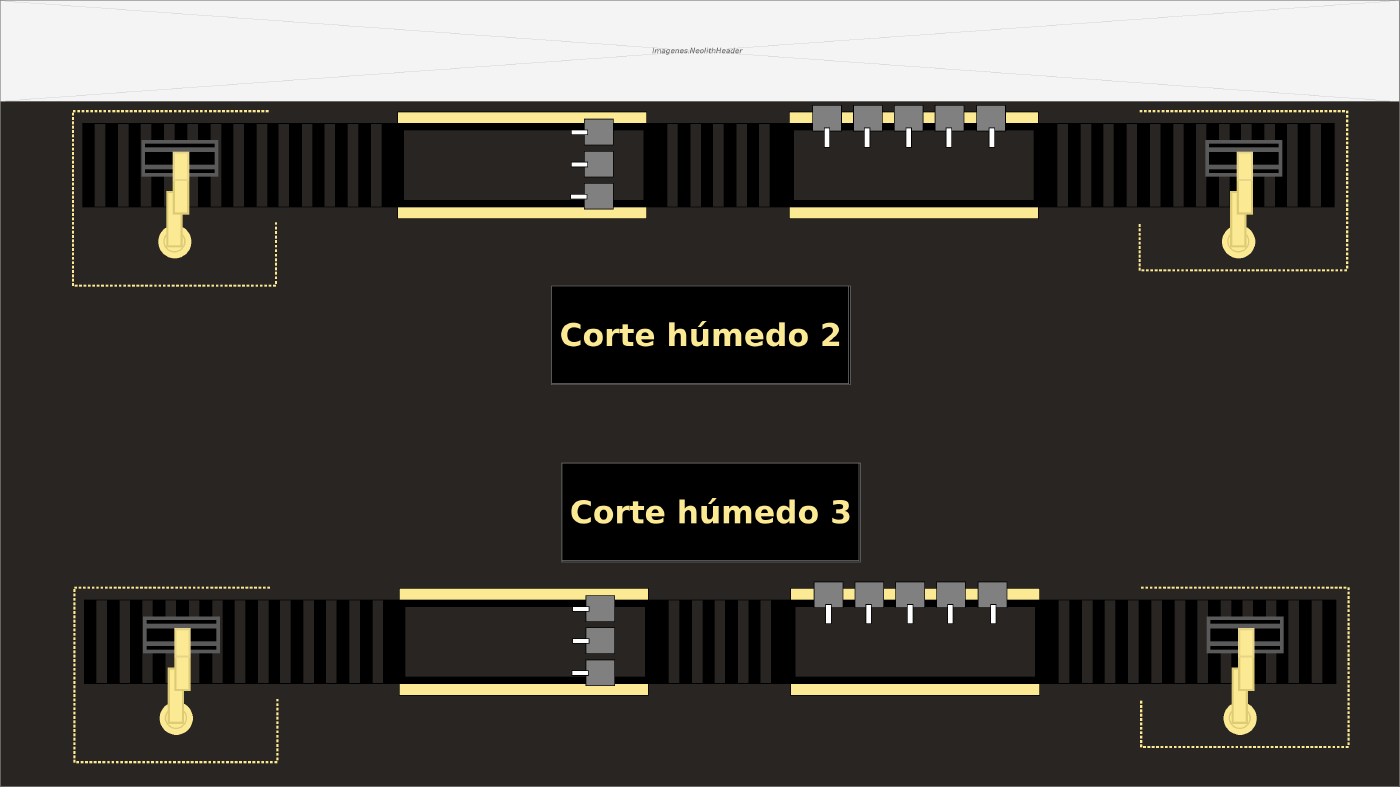
VISUALIZATION Home_Sel_Maq  // 1920x1080
    Button (756,392 410x136), "Corte húmedo 2"
        OnMouseUp: change screen: Home_CortH2
    Button (770,635 410x136), "Corte húmedo 3"
        OnMouseUp: change screen: Home_CortH3
    Image (-7,0 1927x139), image: Imagenes.NeolithHeader
    Group (100,144 1747x248)
        Rectangle (445,9 342x147)
        Rectangle (982,9 342x147)
        Rectangle (13,25 1717x115)
        Group (1349,25 363x115)
            Rectangle (0,0 16x115)
            Rectangle (32,0 16x115)
            Group (63,0 48x115)
                Rectangle (0,0 16x115)
                Rectangle (32,0 16x115)
            Group (127,0 111x115)
                Rectangle (0,0 16x115)
                Rectangle (32,0 16x115)
                Group (63,0 48x115)
                    Rectangle (0,0 16x115)
                    Rectangle (32,0 16x115)
            Rectangle (252,0 16x115)
            Rectangle (284,0 16x115)
            Group (315,0 48x115)
                Rectangle (0,0 16x115)
                Rectangle (32,0 16x115)
        Group (29,25 363x115)
            Rectangle (0,0 16x115)
            Rectangle (32,0 16x115)
            Group (63,0 48x115)
                Rectangle (0,0 16x115)
                Rectangle (32,0 16x115)
            Group (127,0 111x115)
                Rectangle (0,0 16x115)
                Rectangle (32,0 16x115)
                Group (63,0 48x115)
                    Rectangle (0,0 16x115)
                    Rectangle (32,0 16x115)
            Rectangle (252,0 16x115)
            Rectangle (284,0 16x115)
            Group (315,0 48x115)
                Rectangle (0,0 16x115)
                Rectangle (32,0 16x115)
        Rectangle (408,25 16x115)
        Rectangle (453,34 330x97)
        Rectangle (701,19 40x36)
        Rectangle (701,63 40x36)
        Rectangle (701,107 40x36)
        Rectangle (683,34 23x7)
        Rectangle (683,78 23x7)
        Rectangle (682,122 23x7)
        Rectangle (988,34 330x97)
        Rectangle (1014,0 40x36)
        Rectangle (1070,0 40x36)
        Rectangle (1126,0 40x36)
        Rectangle (1182,0 40x36)
        Rectangle (1239,0 40x36)
        Rectangle (1085,31 8x27)
        Rectangle (1030,31 8x27)
        Rectangle (1142,31 8x27)
        Rectangle (1197,31 8x27)
        Rectangle (1256,31 8x27)
        Group (814,25 142x115)
            Rectangle (126,0 16x115)
            Rectangle (0,0 16x115)
            Rectangle (32,0 16x115)
            Group (63,0 48x115)
                Rectangle (0,0 16x115)
                Rectangle (32,0 16x115)
        Polyline (1463,8) (1747,8) (1747,227) (1463,227) (1463,161)
        Polyline (278,161) (278,248) (0,248) (0,8) (271,8)
        Group (94,48 105x162)
            Ellipse (23,117 45x45)
            Ellipse (30,124 30x30)
            RoundedRectangle (34,70 22x77)
            RoundedRectangle (0,0 105x50)
            Rectangle (0,10 105x6)
            Rectangle (0,34 105x6)
            RoundedRectangle (43,25 22x77)
            RoundedRectangle (43,16 22x40)
        Group (1553,48 105x162)
            Ellipse (23,117 45x45)
            Ellipse (30,124 30x30)
            RoundedRectangle (34,70 22x77)
            RoundedRectangle (0,0 105x50)
            Rectangle (0,10 105x6)
            Rectangle (0,34 105x6)
            RoundedRectangle (43,25 22x77)
            RoundedRectangle (43,16 22x40)
    Group (102,798 1747x248)
        Rectangle (445,9 342x147)
        Rectangle (982,9 342x147)
        Rectangle (13,25 1717x115)
        Group (1349,25 363x115)
            Rectangle (0,0 16x115)
            Rectangle (32,0 16x115)
            Group (63,0 48x115)
                Rectangle (0,0 16x115)
                Rectangle (32,0 16x115)
            Group (127,0 111x115)
                Rectangle (0,0 16x115)
                Rectangle (32,0 16x115)
                Group (63,0 48x115)
                    Rectangle (0,0 16x115)
                    Rectangle (32,0 16x115)
            Rectangle (252,0 16x115)
            Rectangle (284,0 16x115)
            Group (315,0 48x115)
                Rectangle (0,0 16x115)
                Rectangle (32,0 16x115)
        Group (29,25 363x115)
            Rectangle (0,0 16x115)
            Rectangle (32,0 16x115)
            Group (63,0 48x115)
                Rectangle (0,0 16x115)
                Rectangle (32,0 16x115)
            Group (127,0 111x115)
                Rectangle (0,0 16x115)
                Rectangle (32,0 16x115)
                Group (63,0 48x115)
                    Rectangle (0,0 16x115)
                    Rectangle (32,0 16x115)
            Rectangle (252,0 16x115)
            Rectangle (284,0 16x115)
            Group (315,0 48x115)
                Rectangle (0,0 16x115)
                Rectangle (32,0 16x115)
        Rectangle (408,25 16x115)
        Rectangle (453,34 330x97)
        Rectangle (701,19 40x36)
        Rectangle (701,63 40x36)
        Rectangle (701,107 40x36)
        Rectangle (683,34 23x7)
        Rectangle (683,78 23x7)
        Rectangle (682,122 23x7)
        Rectangle (988,34 330x97)
        Rectangle (1014,0 40x36)
        Rectangle (1070,0 40x36)
        Rectangle (1126,0 40x36)
        Rectangle (1182,0 40x36)
        Rectangle (1239,0 40x36)
        Rectangle (1085,31 8x27)
        Rectangle (1030,31 8x27)
        Rectangle (1142,31 8x27)
        Rectangle (1197,31 8x27)
        Rectangle (1256,31 8x27)
        Group (814,25 142x115)
            Rectangle (126,0 16x115)
            Rectangle (0,0 16x115)
            Rectangle (32,0 16x115)
            Group (63,0 48x115)
                Rectangle (0,0 16x115)
                Rectangle (32,0 16x115)
        Polyline (1463,8) (1747,8) (1747,227) (1463,227) (1463,161)
        Polyline (278,161) (278,248) (0,248) (0,8) (271,8)
        Group (94,48 105x162)
            Ellipse (23,117 45x45)
            Ellipse (30,124 30x30)
            RoundedRectangle (34,70 22x77)
            RoundedRectangle (0,0 105x50)
            Rectangle (0,10 105x6)
            Rectangle (0,34 105x6)
            RoundedRectangle (43,25 22x77)
            RoundedRectangle (43,16 22x40)
        Group (1553,48 105x162)
            Ellipse (23,117 45x45)
            Ellipse (30,124 30x30)
            RoundedRectangle (34,70 22x77)
            RoundedRectangle (0,0 105x50)
            Rectangle (0,10 105x6)
            Rectangle (0,34 105x6)
            RoundedRectangle (43,25 22x77)
            RoundedRectangle (43,16 22x40)
END_VISUALIZATION

(* stored: Version 1.1.0.1, ProductVersion 3.1.4024.12
   Visu Home_Sel_Maq: Id {5257e64c-3155-462c-b35e-deb33ee21df1} *)
